(* LS Electric XG5000 project: Conveyer_Light_Control_System *)
(* PLC LSPLC *)
(* module base 0 slot 0: FEnet:XGL-EFMT(B) (Fast Ethernet 통신 모듈, 전기 Master) *)
(* module base 0 slot 1: 입력 모듈:XGI-A21A/C (AC 220V 입력, 8점(8점/COM) / 8점(1점/COM)) *)
(* module base 0 slot 2: 출력 모듈:XGQ-RY1A (릴레이 출력, 8점 (2A용, 단독 COM.)) *)

(* Comments on direct variables
%MX3	전체 스위치
%MX4	비상 정지
%MX5	불량 검출
*)

PROGRAM NewProgram (* task: 스캔 프로그램 *)
VAR
    C0 : CTU_INT;
    CV : INT;
    Emergency_Stop AT %IX0.1.1 : BOOL;
    OP_Conveyer AT %QX0.2.5 : BOOL;
    OP_Lamp AT %QX0.2.1 : BOOL;
    OP_Lamp2 AT %QX0.2.2 : BOOL;
    OP_Switch AT %IX0.1.0 : BOOL;
    Search_Defect AT %IX0.1.2 : BOOL;
    T0 : TON;
    T1 : TON;
END_VAR
VAR
    _e1 : R_TRIG;
END_VAR

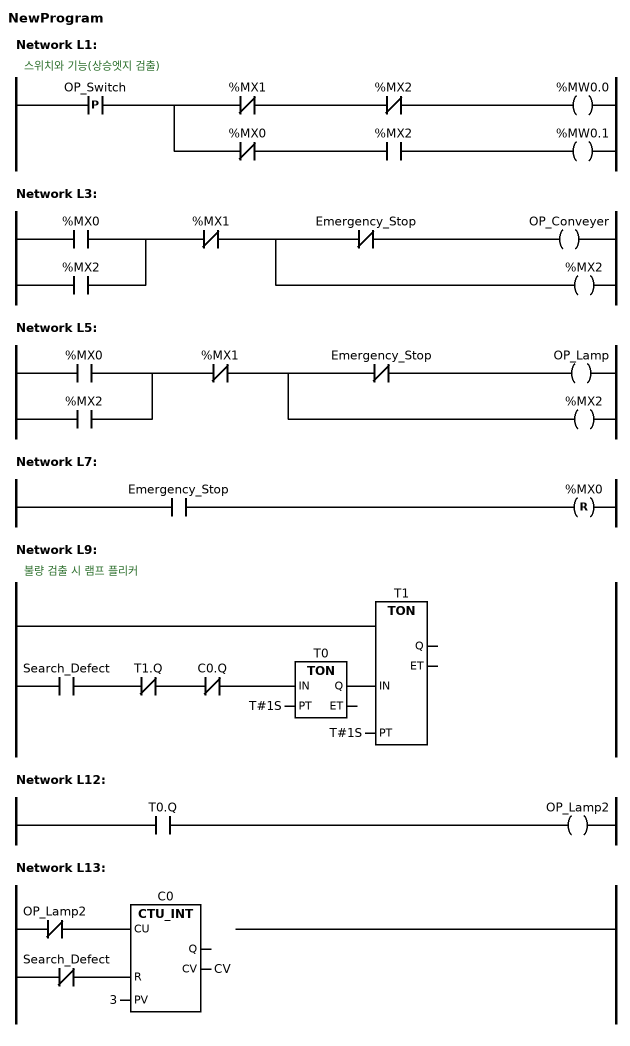
(* 스위치와 기능(상승엣지 검출) *)
(* Rung L1 *)
_e1(CLK := OP_Switch);
%MW0.0 := _e1.Q AND NOT %MX1 AND NOT %MX2;
%MW0.1 := _e1.Q AND NOT %MX0 AND %MX2;
(* Rung L3 *)
OP_Conveyer := (%MX0 OR %MX2) AND NOT %MX1 AND NOT Emergency_Stop;
%MX2 := (%MX0 OR %MX2) AND NOT %MX1;
(* Rung L5 *)
OP_Lamp := (%MX0 OR %MX2) AND NOT %MX1 AND NOT Emergency_Stop;
%MX2 := (%MX0 OR %MX2) AND NOT %MX1;
(* Rung L7 *)
IF Emergency_Stop THEN %MX0 := FALSE; END_IF;
(* 불량 검출 시 램프 플리커 *)
(* Rung L9 *)
T0(IN := Search_Defect AND NOT T1.Q AND NOT C0.Q, PT := T#1S);
T1(IN := T0.Q, PT := T#1S);
(* Rung L12 *)
OP_Lamp2 := T0.Q;
(* Rung L13 *)
C0(CU := NOT OP_Lamp2, R := NOT Search_Defect, PV := 3, CV => CV);
END_PROGRAM

PROGRAM ModbusOnly (* task: 스캔 프로그램 *)
VAR
    C0 : CTU_INT;
    CV : INT;
    Emergency_Stop AT %IX0.1.1 : BOOL;
    OP_Conveyer AT %QX0.2.6 : BOOL;
    OP_Lamp AT %QX0.2.1 : BOOL;
    OP_Lamp2 AT %QX0.2.2 : BOOL;
    OP_Switch AT %IX0.1.0 : BOOL;
    Search_Defect AT %IX0.1.2 : BOOL;
    T0 : TON;
    T1 : TON;
END_VAR
VAR
    _e1 : R_TRIG;
END_VAR

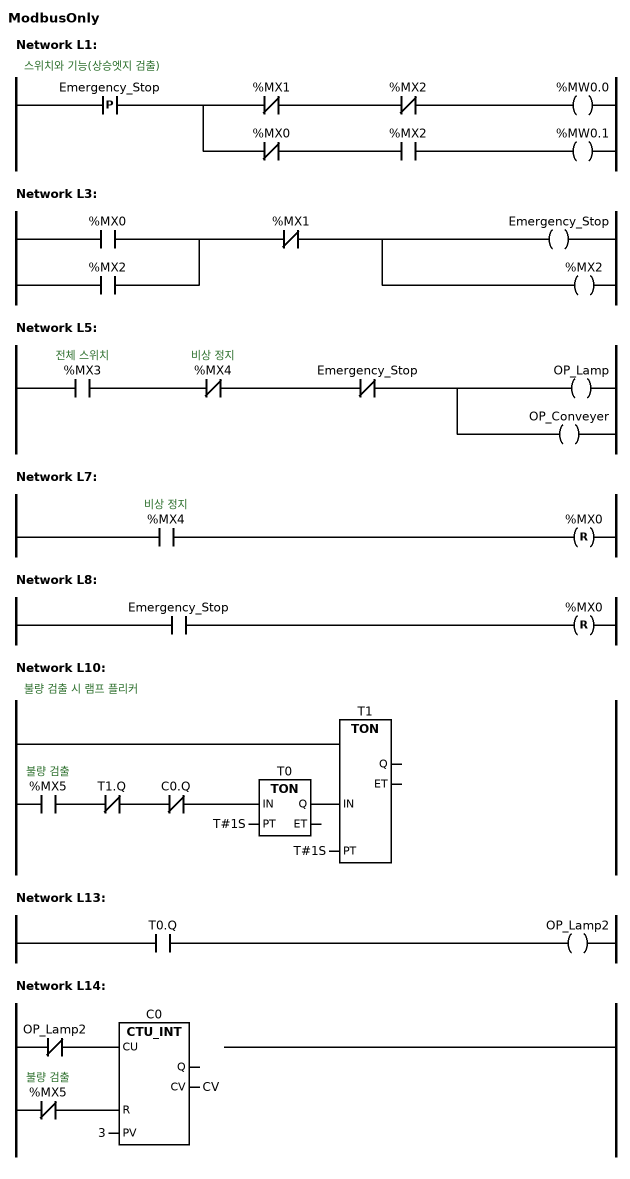
(* 스위치와 기능(상승엣지 검출) *)
(* Rung L1 *)
_e1(CLK := Emergency_Stop);
%MW0.0 := _e1.Q AND NOT %MX1 AND NOT %MX2;
%MW0.1 := _e1.Q AND NOT %MX0 AND %MX2;
(* Rung L3 *)
Emergency_Stop := (%MX0 OR %MX2) AND NOT %MX1;
%MX2 := (%MX0 OR %MX2) AND NOT %MX1;
(* Rung L5 *)
OP_Lamp := %MX3 AND NOT %MX4 AND NOT Emergency_Stop;
OP_Conveyer := %MX3 AND NOT %MX4 AND NOT Emergency_Stop;
(* Rung L7 *)
IF %MX4 THEN %MX0 := FALSE; END_IF;
(* Rung L8 *)
IF Emergency_Stop THEN %MX0 := FALSE; END_IF;
(* 불량 검출 시 램프 플리커 *)
(* Rung L10 *)
T0(IN := %MX5 AND NOT T1.Q AND NOT C0.Q, PT := T#1S);
T1(IN := T0.Q, PT := T#1S);
(* Rung L13 *)
OP_Lamp2 := T0.Q;
(* Rung L14 *)
C0(CU := NOT OP_Lamp2, R := NOT %MX5, PV := 3, CV => CV);
END_PROGRAM